PROGRAM P_Demo_FB_JsonDomParser_PushbackStringValue
VAR
    fbParser : FB_JsonDomParser; // 父 FB 实例
    v : SJsonValue;
    value : STRING(255);
    vRet : SJsonValue; // 返回值监视
    bTrigger : BOOL := FALSE; // 在线置 TRUE 触发一次调用
    bTriggerPrev : BOOL;
END_VAR

// =============================================================================
// 场景：循环把采样数据加入 JSON 数组（如 1 秒采 10 次温度，组成 10 元素数组上报）。
// 价值：按位 append 比每次重建数组高效。
// 验证：登录 PLC 在线写 bTrigger := TRUE 触发，monitor 返回值/输出参数。具体步骤见下方注释。
// 验证步骤：
//   1. 右键 PLC 项目下 POUs 文件夹 → Add → Existing Item → 选本 .TcPOU 文件
//   2. 引用 Tc3_JsonXml（References → Add library）
//   3. 编译 → 登录 → 运行；按 verify 注释里给出的在线写值操作
// =============================================================================

// 上升沿触发一次方法调用并观察输出。
IF bTrigger AND NOT bTriggerPrev THEN
    vRet := fbParser.PushbackStringValue(
        v := v,
        value := value
    );
END_IF;
bTriggerPrev := bTrigger;

END_PROGRAM

(* stored: Version 1.1.0.1, ProductVersion 3.1.4024.5
   POU P_Demo_FB_JsonDomParser_PushbackStringValue: Id {45fb8c91-ff15-5c39-856f-5101e16528a5}, SpecialFunc None *)
